INTERFACE I_NodeAddedEvent EXTENDS I_Event

PROPERTY PUBLIC Target : I_Node
GET
END_GET
END_PROPERTY

END_INTERFACE

(* stored: Version 1.1.0.1, ProductVersion 3.1.4024.12
   Itf I_NodeAddedEvent: Id {b49ed444-70a6-4f21-b512-54d181da37ff}
   Property Target: Id {4087ad35-7496-4252-ae90-a07fa752a36a}
   Get Get: Id {6d7040ff-3f2d-4f9c-96fb-ead839040719} *)
